{attribute addProperty BoxType "EL2521-0000-1016"}
{attribute addProperty Id "Sel_Ack_End_counterAT %I*BOOL811Ramp_activeAT %I*BOOL812Status_of_input_targetAT %I*BOOL815Status_of_input_zeroAT %I*BOOL816ErrorAT %I*BOOL817Sync_ErrorAT %I*BOOL8132TxPDO_ToggleAT %I*BOOL819"}
{attribute addProperty CRC "3407757998"}
{attribute addProperty SizeInBites "56"}
{attribute addProperty SizeInBytes "7"}
TYPE PTO_Status_CB1E42AE :
STRUCT
	{attribute addProperty Name "Sel_Ack_End_counter"}
	Sel_Ack_End_counter AT %I* : BOOL;
	{attribute addProperty Name "Ramp_active"}
	Ramp_active AT %I* : BOOL;
	{attribute addProperty Name "Status_of_input_target"}
	Status_of_input_target AT %I* : BOOL;
	{attribute addProperty Name "Status_of_input_zero"}
	Status_of_input_zero AT %I* : BOOL;
	{attribute addProperty Name "Error"}
	Error AT %I* : BOOL;
	{attribute addProperty Name "Sync_Error"}
	Sync_Error AT %I* : BOOL;
	{attribute addProperty Name "TxPDO_Toggle"}
	TxPDO_Toggle AT %I* : BOOL;
END_STRUCT
END_TYPE

(* stored: Version 1.2.0.0, ProductVersion 3.1.4024.9
   DUT PTO_Status_CB1E42AE: Id {33e10177-93d2-40dd-9a47-36470fa1a33f} *)
